Staubli VAL3: splitStr.pgx

program split(string x_sSourceStr, string& x_sDestStr[])
  local string l_sSplitChar[3]
  local num l_nX
  local num l_nCount
  local num l_nFirstIndex
  local num l_nMaxIndex
  local num l_nBuffIndex
begin
  //



  //参数初始化
  l_sSplitChar[0]="/"
  l_sSplitChar[1]=","
  l_sSplitChar[2]="="



  for l_nX=0 to size(x_sDestStr,1)-1
    x_sDestStr[l_nX]=""
  endFor


  //参数合法化判断
  if x_sSourceStr==""
    return
  endIf


  //进行分解
  while true

    l_nMaxIndex=-2000
    l_nFirstIndex=2000

    //判断值
    for l_nX=0 to size(l_sSplitChar,1)-1
      l_nBuffIndex=find(x_sSourceStr,l_sSplitChar[l_nX])
      l_nMaxIndex=max(l_nMaxIndex,l_nBuffIndex)
      if l_nBuffIndex<l_nFirstIndex and l_nBuffIndex>=0
        l_nFirstIndex=l_nBuffIndex
      endIf
    endFor


    //退出
    if l_nMaxIndex<0 or l_nCount>=size(x_sDestStr,1)-1
      x_sDestStr[l_nCount]=x_sSourceStr
      return
    endIf



    //分割
    x_sDestStr[l_nCount]=left(x_sSourceStr,l_nFirstIndex)
    x_sSourceStr=right(x_sSourceStr,len(x_sSourceStr)-l_nFirstIndex-1)

    l_nCount=l_nCount+1


  endWhile



end
